RoboDK station: simulation_broken.rdk

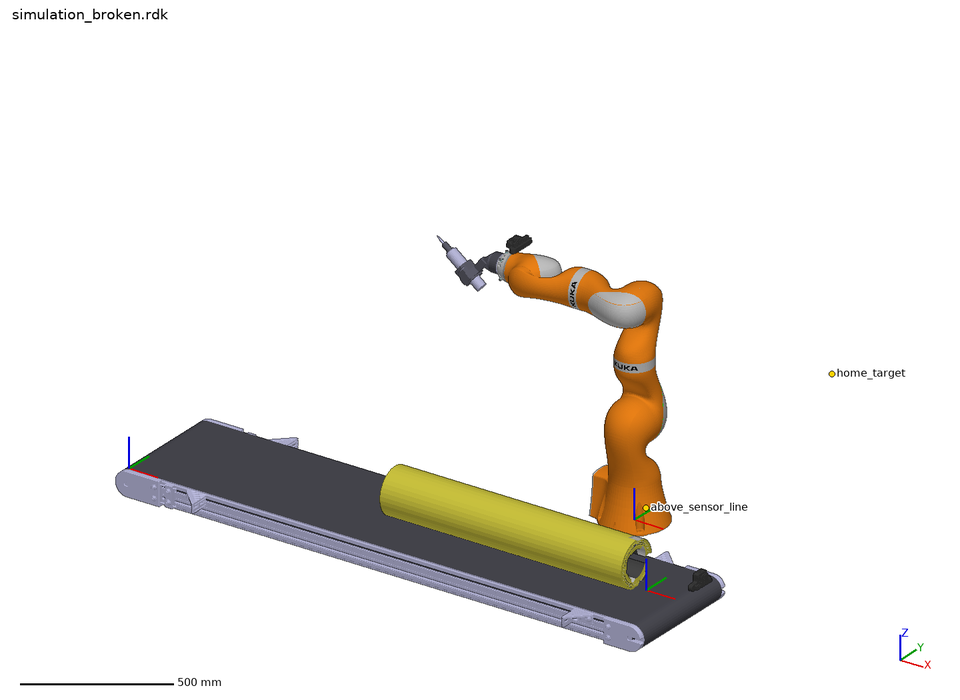
[picture v0: the station drawn from its stored meshes, robots at their saved joint values, targets as dots, program paths as lines]
Station simulation (saved by RoboDK 5.5.1). Poses are relative to the parent item; angles as X-Y-Z fixed-axis rotations.
  - frame Conveyor Belt (2m) Base at (0, 0, 0) mm
    - robot Conveyor: 1 axes
        modified DH rows (alpha deg, a mm, theta deg, d mm): 0, 0, 0, 0 linear
        base shift (0, 0, 0) mm, rotated rx 0 ry 90 rz 0 deg
        joint limits [-500000] to [500000]; home [0]; saved at [1900]
      - frame Conveyor Object at (0, 225, 0) mm
        - object pipe at (0, -87, 0) mm, rotated rx 0 ry -90 rz 0 deg, size 173.7 x 173.8 x 960 mm, geometry from pipe.STL
        - object pipe_broken at (-1000, -87, 172) mm, rotated rx 0 ry 90 rz 0 deg, size 174 x 173.8 x 960 mm, geometry from pipe_broken.STL
    - target conveyor_home (joint target) at (0, 0, 0) mm; joints [0] of Conveyor
    - target conveyor_end (Cartesian target) at (2000, 0, 0) mm; joints [2000] of Conveyor
  - camera side_camera
  - object side_cam at (1400, 225, 1100) mm, rotated rx 180 ry 0 rz 90 deg, size 110 x 54.5 x 33 mm, geometry from OpenCV-OAK-D-Camera.sld
  - object section_cam at (2100, 225, 87) mm, rotated rx -90 ry 0 rz 90 deg, size 110 x 54.5 x 33 mm, geometry from OpenCV-OAK-D-Camera.sld
  - camera section_camera
  - frame KUKA LBR iiwa 14 R820 Base at (1450, 800, -100) mm
    - robot KUKA LBR iiwa 14 R820: 7 axes, payload 14 kg, reach 820 mm, repeatability 0.1 mm, weight 29.9 kg
        modified DH rows (alpha deg, a mm, theta deg, d mm): 0, 0, 0, 360; -90, 0, 0, 0; 90, 0, 0, 420; -90, 0, 0, 0; 90, 0, 0, 400; -90, 0, 0, 0; 90, 0, 0, 126
        joint limits [-170, -120, -170, -120, -170, -120, -175] to [170, 120, 170, 120, 170, 120, 175]; home [0, 0, 0, -90, 0, 0, 0]; saved at [0, 0, 0, -90, 0, 0, 0]
      - tool Spindle, TCP at (32, 0, 260) mm, rotated rx 0 ry 39 rz 0 deg, size 157.3 x 72 x 259.9 mm
    - target above_sensor_line (Cartesian target) at (450, -575, 400) mm, rotated rx 180 ry 0 rz 90 deg; joints [-38.422, 24.62, 0, -68.49, -33.154, 64.362, 60.196] of KUKA LBR iiwa 14 R820
    - target home_target (Cartesian target) at (786, 0, 748) mm, rotated rx 180 ry 51 rz 180 deg; joints [0, 0, 0, -90, 0, 0, 0] of KUKA LBR iiwa 14 R820
  - Python program main (listed below)

--- Python program main ---
from robodk import robolink    # RoboDK API
from robodk import robomath    # Robot toolbox
from robodk.robomath import *

import sys

# caution: path[0] is reserved for script path (or '' in REPL)
sys.path.insert(1, 'D:\pipe_repo\pipe-recognisation\robotic_simulation')
sys.path.insert(2, 'INSERT YOUR PATH HERE TO THE robotic_simulation FOLDER')

from python_files.object_measurement import object_measurement
from python_files.layer_segmentation import layer_segmentation
from python_files.operate_side_cam import get_side_cam
from python_files.init_cams import init_cams
from python_files.init_conv_pos import init_conv_pos
from python_files.move_conv import move_conv
from python_files.operate_section_cam import get_section_cam
from python_files.robot_move_dimensions import robot_move_dimensions
from python_files.robot_move_layers import robot_move_layers
from python_files.get_dimensions import get_dimensions
from python_files.get_layers import get_layers
from python_files.init_robot import init_robot

import numpy as np
import cv2
RDK = robolink.Robolink()
SIDE_CAM_HEIGHT = 1.1
SIDE_CAM_FOV = 60
SECTION_CAM_DIS = 0.2
SECTION_CAM_FOV = 60

init_robot()
init_cams()
init_conv_pos()
move_conv()
image_side = get_side_cam()
image_section = get_section_cam()
dimension_image, length, side_diameter = get_dimensions(image_side, SIDE_CAM_HEIGHT, SIDE_CAM_FOV)
layers_image, radii = get_layers(image_section, SECTION_CAM_DIS, SECTION_CAM_FOV)
section_diameter = radii[-1]*2
avg_diameter = (section_diameter + side_diameter)/2


cv2.imshow("dim", dimension_image)
cv2.imshow("layers", layers_image)
cv2.waitKey(0) # PRESS A KEY ON THE IMAGES WINDOW TO CONTINUE
cv2.destroyAllWindows()

robot_move_dimensions(length, avg_diameter)
robot_move_layers(radii)
